(*
SPDX-FileCopyrightText: © 2026 Oleksandr Tiutyk <trofimich@gmail.com>
SPDX-License-Identifier: MIT
License: https://opensource.org/license/mit
*)

(*!
<summary>Suppresses test log output and optionally simulates reuse of a native diagnostic during logging.</summary>
<description>Probe state belongs to the calling cyclic task. The filter never retains the borrowed exception.</description>
*)

{attribute 'no_explicit_call' := 'do not call this function block directly'}
FUNCTION_BLOCK LogFilter EXTENDS TOF_Core.Object IMPLEMENTS TOF_Core.ILogFilter
VAR
	_SecondaryExceptionPending : ARRAY [1..TOF_Core.System.TASK_COUNT] OF BOOL;
END_VAR
VAR_STAT
	//! <summary>Class name shared by all instances of this function block.</summary>
	{attribute 'hide'} 
	_ClassName : STRING := __POUNAME();
END_VAR

{attribute 'monitoring' := 'call'}
PROPERTY ClassName : REFERENCE TO STRING
GET
ClassName REF= _ClassName;
END_GET
END_PROPERTY

{attribute 'monitoring' := 'call'}
PROPERTY NamespaceName : REFERENCE TO STRING
GET
NamespaceName REF= CurrentNamespace.Name;
END_GET
END_PROPERTY

{attribute 'monitoring' := 'call'}
PROPERTY SelfSize : ULINT
GET
SelfSize := XSIZEOF(THIS^);
END_GET
END_PROPERTY

(*! <summary>Consumes any armed secondary diagnostic in this task and suppresses the log entry.</summary> *)
METHOD ShouldLog : BOOL
VAR_IN_OUT CONSTANT
	category : TOF_Core.LOG_CATEGORY;
	topics : ARRAY [*] OF WSTRING;		
END_VAR
VAR
	taskIndex : DINT;
END_VAR
taskIndex := TOF_Core.System.GetCurrentTaskIndex();

IF taskIndex >= 1
	AND_THEN taskIndex <= TOF_Core.System.TASK_COUNT
	AND_THEN _SecondaryExceptionPending[taskIndex]
THEN
	_SecondaryExceptionPending[taskIndex] := FALSE;
	TOF_Core.ExceptionManager.GetLastException(
		exceptionCode := __SYSTEM.ExceptionCode.RTSEXCPT_ACCESS_VIOLATION,
		catchPointNamespaceName := NamespaceName,
		catchPointPOUName := __POUNAME(),
		catchPointPosition := __POSITION()
	);
END_IF

ShouldLog := FALSE;
END_METHOD

(*!
<summary>Enables or cancels one simulated secondary native diagnostic in the calling test task.</summary>
<description>Each cyclic task owns its slot. Other tasks keep their configured filter behavior.</description>
<param name="enabled">TRUE arms the next logging callback. FALSE cancels a pending probe.</param>
*)
METHOD SetSecondaryExceptionProbe
VAR_INPUT
	enabled : BOOL;
END_VAR
VAR
	taskIndex : DINT;
END_VAR
taskIndex := TOF_Core.System.GetCurrentTaskIndex();

IF taskIndex >= 1 AND_THEN taskIndex <= TOF_Core.System.TASK_COUNT THEN
	_SecondaryExceptionPending[taskIndex] := enabled;
END_IF
END_METHOD

END_FUNCTION_BLOCK

(* stored: Version 1.1.0.1, ProductVersion 3.1.4026.21
   POU LogFilter: Id {a3a9bf30-d5a5-47cf-b4ee-55ca6a681ea6}, SpecialFunc None
   Property ClassName: Id {cae48fd3-c4fa-4ca2-868f-5de6218356a4}
   Get Get: Id {0975c72d-6209-4578-829a-a4591272bc5e}
   Property NamespaceName: Id {68024585-ccb0-40a1-b903-f0eeb9d6b824}
   Get Get: Id {2aec628d-2163-4d74-b6e4-af288f4660b2}
   Property SelfSize: Id {85c32638-abaa-4f8a-acf0-0653e4aebcdd}
   Get Get: Id {8e3c09a4-76e1-4529-a461-2e5e2464bde1}
   Method ShouldLog: Id {32b9de1c-02d2-47a5-837f-c1e69ba1998b}
   Method SetSecondaryExceptionProbe: Id {923620dc-252b-43bf-ab55-0111d4df69a4} *)
